SUBAPPLICATION Uebung_033 (* LED Strip Blinkende LED *)
  (* Standard: 61499-2; Description: Copyright (c) 2023 Meisterschulen am Ostbahnhof This program and the accompanying materials are made available under the terms of the Eclipse Public License 2.0 which is available at https://www.eclipse.org/legal/epl-2.0/ SPDX-License-Identifier: EPL-2.0 *)
  (* Version 1.0, 2023-10-23, Franz Höpfinger, Meisterschulen am Ostbahnhof *)
  PACKAGE Uebungen;
  IMPORT logiBUS::io::DI::logiBUS_DI::Input_I1;
  IMPORT logiBUS::io::DI::logiBUS_DI::Input_I2;
  IMPORT logiBUS::io::DI::logiBUS_DI::Input_I3;
  IMPORT logiBUS::io::DI::logiBUS_DI::Input_I4;
  IMPORT logiBUS::io::DO_LED::LED_COLOURS;
  IMPORT logiBUS::io::DO_LED::LED_strip;
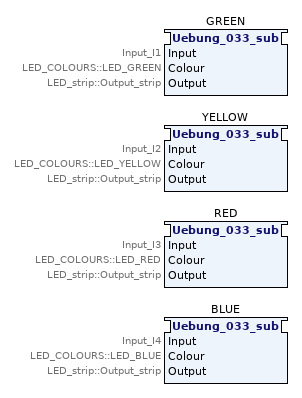
  SUBAPPS
    GREEN : Uebungen::Uebung_033_sub(Input := Input_I1, Colour := LED_COLOURS::LED_GREEN, Output := LED_strip::Output_strip);
    YELLOW : Uebungen::Uebung_033_sub(Input := Input_I2, Colour := LED_COLOURS::LED_YELLOW, Output := LED_strip::Output_strip);
    RED : Uebungen::Uebung_033_sub(Input := Input_I3, Colour := LED_COLOURS::LED_RED, Output := LED_strip::Output_strip);
    BLUE : Uebungen::Uebung_033_sub(Input := Input_I4, Colour := LED_COLOURS::LED_BLUE, Output := LED_strip::Output_strip);
  END_SUBAPPS
END_SUBAPPLICATION
